(* IEC 61131-3 sources: std_i2980_v2.06_cp053/Source/IMM/ieccontrol/MoldGeneral (part 4) *)

(* ---- ABManualButton.pu ---- *)
(*
@h    ! WARNING !
@h    The Kemro K2 system (including software) only meets category B according to EN 954-1,
@h    thus it is not intended for usage in safety-relevant control applications in the field
@h    of personal safety (e.g. emergency stop).
@h    To implement potentially necessary safety-relevant control tasks, always use additional
@h    external safety devices that are intended for the particular purpose, and meet the necessary
@h    functional safety.
@h    For further information see EN 954-1 (EN ISO 13849-1) and/or the K2-x00 user manual, chapter
@h    "CE conformity, directives and standards".

react to manual buttons
find next target position when button is pressed

@FunctionID: S_FU_01_Mold1
*)

IMPORT_OVER_LISTFILE
 IS_LINKED
, cMoveFwd
, cMoveBwd
, cCompMoldHeightAuto
, cMoveBwdInterPos
, FBManualButton
, tsDeviceId
, tsInterCondList
, tsMoveData
, tyInstanceListArray
, tyInterCondBoolArray
, tMoveIdent
, FBCheckReady

END_IMPORT

ALGORITHM_BLOCK ABManualButton #DUMMY_EDIT_BLOCK

SYSTEM_VAR
 sv_bInitDone : BOOL;
 sv_DeviceId : tsDeviceId;
 sv_rMoldPosition : REAL;
 sv_FwdInterruptList : tsInterCondList (* list with interrupt positions for mold close *);
 sv_BwdInterruptList : tsInterCondList (* list with interrupt positions for mold open *);
 sv_MoveCloseInterPos : tsMoveData;
 sv_MoveOpenInterPos : tsMoveData;
 sv_bUseProgramSwitches : BOOL;
 sv_InstanceDataCloseInterPos : tyInstanceListArray;
 sv_InstanceDataOpenInterPos : tyInstanceListArray;
 sv_CloseInterPosProgInSequ : tyInterCondBoolArray (* information, which instances of mold close interpos movement are programmed in sequence  *);
 sv_OpenInterPosProgInSequ : tyInterCondBoolArray (* information, which instances of mold open interpos movement are programmed in sequence *);
END_VAR

SYSTEM_OBJECT
 PU_Task_7 : TASK;
END_OBJECT

VAR
 fbManualButton : FBManualButton;
 mpbAutoAdjustReady : REFTO BOOL;
END_VAR

ALGORITHM aGetNextCloseMovement

VAR_OUTPUT
 MoveId : tMoveIdent;
 iInstance : DINT;
END_VAR

VAR_TEMP
 i : DINT;
END_VAR
#BEGIN_EDIT_BLOCK
(**************************************** WARNING ********************************************
 *** The KEBA Kemro K2 System including software is not intended for safety control tasks! ***
 ***                       For further information see Comment tab!                        ***
 *********************************************************************************************)

MoveId := cMoveFwd;
iInstance := 1;

IF sv_bUseProgramSwitches THEN
   //get next target position from sv_FwdInterruptList
   FOR i := 1 TO sv_FwdInterruptList.iUsedElements DO
      IF (sv_FwdInterruptList.List[i].rTargetValue < sv_rMoldPosition) THEN
         iInstance := i;
         MoveId := cMoveFwdInterPos;
         RETURN;
      END_IF;
   END_FOR;
ELSE
   //sequence programmed by editor
   //-> check instance data to get next target position
   FOR i := 1 TO cMaxIntermediateConditions DO
      IF sv_CloseInterPosProgInSequ[i] AND sv_InstanceDataCloseInterPos[i].rTargetValue < sv_rMoldPosition THEN
         iInstance := i;
         MoveId := cMoveFwdInterPos;
         RETURN;
      END_IF;
   END_FOR;
END_IF;

;#END_EDIT_BLOCK END_ALGORITHM

ALGORITHM aGetNextOpenMovement

VAR_OUTPUT
 MoveId : tMoveIdent;
 iInstance : DINT;
END_VAR

VAR_TEMP
 i : DINT;
END_VAR
#BEGIN_EDIT_BLOCK
(**************************************** WARNING ********************************************
 *** The KEBA Kemro K2 System including software is not intended for safety control tasks! ***
 ***                       For further information see Comment tab!                        ***
 *********************************************************************************************)

MoveId := cMoveBwd;
iInstance := 1;

IF sv_bUseProgramSwitches THEN
   //get next target position from sv_BwdInterruptList
   FOR i := 1 TO sv_BwdInterruptList.iUsedElements DO
      IF (sv_BwdInterruptList.List[i].rTargetValue > sv_rMoldPosition) THEN
         iInstance := i;
         MoveId := cMoveBwdInterPos;
         RETURN;
      END_IF;
   END_FOR;
ELSE
   //sequence programmed by editor
   //-> check instance data to get next target position
   FOR i := 1 TO cMaxIntermediateConditions DO
      IF sv_OpenInterPosProgInSequ[i] AND sv_InstanceDataOpenInterPos[i].rTargetValue > sv_rMoldPosition THEN
         iInstance := i;
         MoveId := cMoveBwdInterPos;
         RETURN;
      END_IF;
   END_FOR;
END_IF;

;#END_EDIT_BLOCK END_ALGORITHM

ALGORITHM aButtonClose

VAR_INPUT
 bButtonClose : BOOL;
END_VAR

VAR
 MoveId : tMoveIdent;
 iIntermediateCond : DINT;
END_VAR
#BEGIN_EDIT_BLOCK
(**************************************** WARNING ********************************************
 *** The KEBA Kemro K2 System including software is not intended for safety control tasks! ***
 ***                       For further information see Comment tab!                        ***
 *********************************************************************************************)

IF mpbAutoAdjustReady <> EMPTY AND NOT mpbAutoAdjustReady^ THEN
    // auto mold adjust available and active -> ignore manual button
    RETURN;
END_IF;

IF bButtonClose THEN

   IF sv_MoveCloseInterPos.bProgrammedInSequence THEN
      //mold close movement to interpos programmed in sequence
      aGetNextCloseMovement(MoveId => MoveId,
                            iInstance => iIntermediateCond);
   ELSE
      //no interpos movement programmed
      MoveId := cMoveFwd;
      iIntermediateCond := 1;
   END_IF;

END_IF;

fbManualButton(bButton := bButtonClose, MoveId := MoveId, MoveDir := cMoveFwd, IntermediateCond := iIntermediateCond);

;#END_EDIT_BLOCK END_ALGORITHM

ALGORITHM aButtonOpen

VAR_INPUT
 bButtonOpen : BOOL;
END_VAR

VAR
 MoveId : tMoveIdent;
 iIntermediateCond : DINT;
END_VAR
#BEGIN_EDIT_BLOCK
(**************************************** WARNING ********************************************
 *** The KEBA Kemro K2 System including software is not intended for safety control tasks! ***
 ***                       For further information see Comment tab!                        ***
 *********************************************************************************************)

IF mpbAutoAdjustReady <> EMPTY AND NOT mpbAutoAdjustReady^ THEN
    // auto mold adjust available and active -> ignore manual button
    RETURN;
END_IF;

IF bButtonOpen THEN

   IF sv_MoveOpenInterPos.bProgrammedInSequence THEN
      //mold open movement to interpos programmed in sequence
      aGetNextOpenMovement(MoveId => MoveId,
                           iInstance => iIntermediateCond);
   ELSE
      //no interpos movement programmed
      MoveId := cMoveBwd;
      iIntermediateCond := 1;
   END_IF;

END_IF;

fbManualButton(bButton := bButtonOpen, MoveId := MoveId, MoveDir := cMoveBwd, IntermediateCond := iIntermediateCond);

;#END_EDIT_BLOCK END_ALGORITHM

POSTUPDATE_ALGORITHM pInitDone ON PU_Task_7(10) WITH sv_bInitDone

VAR
 fbCheckAutoAdjustReady : FBCheckReady;
 DeviceIdAutoAdjust : tsDeviceId;
END_VAR
#BEGIN_EDIT_BLOCK
(**************************************** WARNING ********************************************
 *** The KEBA Kemro K2 System including software is not intended for safety control tasks! ***
 ***                       For further information see Comment tab!                        ***
 *********************************************************************************************)

//get reference to ready flag of auto mold adjust function unit
DeviceIdAutoAdjust.CompId := cCompMoldHeightAuto;
DeviceIdAutoAdjust.IndexId := sv_DeviceId.IndexId;

fbCheckAutoAdjustReady(DeviceId := DeviceIdAutoAdjust);
mpbAutoAdjustReady := fbCheckAutoAdjustReady.pbReady;

;#END_EDIT_BLOCK END_ALGORITHM

END_ALGORITHM_BLOCK

#END_OF_IEC_PART

@Puma @IecEditor 6 97 @Pou 25
@@@BEG_Comment@@@
@h    ! WARNING !
@h    The Kemro K2 system (including software) only meets category B according to EN 954-1,
@h    thus it is not intended for usage in safety-relevant control applications in the field
@h    of personal safety (e.g. emergency stop).
@h    To implement potentially necessary safety-relevant control tasks, always use additional
@h    external safety devices that are intended for the particular purpose, and meet the necessary
@h    functional safety.
@h    For further information see EN 954-1 (EN ISO 13849-1) and/or the K2-x00 user manual, chapter
@h    "CE conformity, directives and standards".

react to manual buttons
find next target position when button is pressed

@FunctionID: S_FU_01_Mold1
@@@END_Comment@@@

@BEG_Contents

@BEG_Func
@RT(17)FuncTreeContainer
1
@Var @RT(9)IS_LINKED @RT(0) @T @T @DERIVED 0 @F @RT(22)KEBA_STANDARD_FUNCTION @F
@T
@BEG_Attrib
0 @RT(0) @RT(0)
@END_Attrib
1 1 @F @F @F @F

@END_Func

@BEG_Const
@RT(18)ConstTreeContainer
4
@Var @RT(8)cMoveFwd @RT(0) @T @F @DT @RT(4)DINT @RT(0) @T @T @BASIC 0 @F
@F @F
@T
@BEG_Attrib
0 @RT(2)12 @RT(16)movement forward
@END_Attrib
1 1 @F @F @F @F

@Var @RT(8)cMoveBwd @RT(0) @T @F @DT @RT(4)DINT @RT(0) @T @T @BASIC 0 @F
@F @F
@T
@BEG_Attrib
0 @RT(2)11 @RT(17)movement backward
@END_Attrib
1 1 @F @F @F @F

@Var @RT(19)cCompMoldHeightAuto @RT(0) @T @F @DT @RT(4)DINT @RT(0) @T @T @BASIC 0 @F
@F @F
@T
@BEG_Attrib
0 @RT(3)125 @RT(26)Component Auto Mold Height
@END_Attrib
1 1 @F @F @F @F

@Var @RT(16)cMoveBwdInterPos @RT(0) @T @F @DT @RT(4)DINT @RT(0) @T @T @BASIC 0 @F
@F @F
@T
@BEG_Attrib
0 @RT(2)16 @RT(38)move backward to intermediate position
@END_Attrib
1 1 @F @F @F @F

@END_Const

@BEG_Export

@BEG_Kind
@ALGORITHM_BLOCK @RT(14)ABManualButton @STRUCTURED_TEXT
@RT(0) @RT(0) @RT(0)
@END_Kind

@BEG_Dcl
@RT(16)DclTreeContainer
15
@Var @RT(9)PU_Task_7 @RT(0) @T @T @RENAMED 0 @T @T @DT @RT(4)TASK @RT(0) @T @T @BASIC 0 @F
@F @F
@T
@BEG_Attrib
3 @RT(0) @RT(0) @RT(0)
@END_Attrib
1 7 @F @F @F @F

@Var @RT(14)fbManualButton @RT(0) @T @T @DERIVED 0 @T @T @DT @RT(14)FBManualButton @RT(0) @T @T @UNKNOWN 0 @F
@F @F
@T
@BEG_Attrib
3 @RT(0) @RT(0) @RT(0)
@END_Attrib
1 0 @F @F @F @F

@Var @RT(12)sv_bInitDone @RT(0) @T @F @DT @RT(4)BOOL @RT(0) @T @T @BASIC 0 @F
@F @F
@T
@BEG_Attrib
3 @RT(0) @RT(0) @RT(0)
@END_Attrib
1 8 @F @F @F @F

@Var @RT(11)sv_DeviceId @RT(0) @T @T @DERIVED 0 @T @T @DT @RT(10)tsDeviceId @RT(0) @T @T @UNKNOWN 0 @F
@F @F
@T
@BEG_Attrib
3 @RT(0) @RT(0) @RT(0)
@END_Attrib
1 8 @F @F @F @F

@Var @RT(18)mpbAutoAdjustReady @RT(0) @T @T @REFTO 0 @T @DT @RT(4)BOOL @RT(0) @T @T @BASIC 0 @F
@F @F
@T
@BEG_Attrib
3 @RT(0) @RT(0) @RT(0)
@END_Attrib
1 0 @F @F @F @F

@Var @RT(16)sv_rMoldPosition @RT(0) @T @F @DT @RT(4)REAL @RT(0) @T @T @BASIC 0 @F
@F @F
@T
@BEG_Attrib
3 @RT(0) @RT(0) @RT(0)
@END_Attrib
1 8 @F @F @F @F

@Var @RT(19)sv_FwdInterruptList @RT(0) @T @T @DERIVED 0 @T @T @DT @RT(15)tsInterCondList @RT(0) @T @T @UNKNOWN 0 @F
@F @F
@T
@BEG_Attrib
3 @RT(0) @RT(44)list with interrupt positions for mold close @RT(0)
@END_Attrib
1 8 @F @F @F @F

@Var @RT(19)sv_BwdInterruptList @RT(0) @T @T @DERIVED 0 @T @T @DT @RT(15)tsInterCondList @RT(0) @T @T @UNKNOWN 0 @F
@F @F
@T
@BEG_Attrib
3 @RT(0) @RT(43)list with interrupt positions for mold open @RT(0)
@END_Attrib
1 8 @F @F @F @F

@Var @RT(20)sv_MoveCloseInterPos @RT(0) @T @T @DERIVED 0 @T @T @DT @RT(10)tsMoveData @RT(0) @T @T @UNKNOWN 0 @F
@F @F
@T
@BEG_Attrib
3 @RT(0) @RT(0) @RT(0)
@END_Attrib
1 8 @F @F @F @F

@Var @RT(19)sv_MoveOpenInterPos @RT(0) @T @T @DERIVED 0 @T @T @DT @RT(10)tsMoveData @RT(0) @T @T @UNKNOWN 0 @F
@F @F
@T
@BEG_Attrib
3 @RT(0) @RT(0) @RT(0)
@END_Attrib
1 8 @F @F @F @F

@Var @RT(22)sv_bUseProgramSwitches @RT(0) @T @F @DT @RT(4)BOOL @RT(0) @T @T @BASIC 0 @F
@F @F
@T
@BEG_Attrib
3 @RT(0) @RT(0) @RT(0)
@END_Attrib
1 8 @F @F @F @F

@Var @RT(28)sv_InstanceDataCloseInterPos @RT(0) @T @T @DERIVED 0 @T @T @DT @RT(19)tyInstanceListArray @RT(0) @T @T @UNKNOWN 0 @F
@F @F
@T
@BEG_Attrib
3 @RT(0) @RT(0) @RT(0)
@END_Attrib
1 8 @F @F @F @F

@Var @RT(27)sv_InstanceDataOpenInterPos @RT(0) @T @T @DERIVED 0 @T @T @DT @RT(19)tyInstanceListArray @RT(0) @T @T @UNKNOWN 0 @F
@F @F
@T
@BEG_Attrib
3 @RT(0) @RT(0) @RT(0)
@END_Attrib
1 8 @F @F @F @F

@Var @RT(26)sv_CloseInterPosProgInSequ @RT(0) @T @T @DERIVED 0 @T @T @DT @RT(20)tyInterCondBoolArray @RT(0) @T @T @UNKNOWN 0 @F
@F @F
@T
@BEG_Attrib
3 @RT(0) @RT(88)information, which instances of mold close interpos movement are programmed in sequence  @RT(0)
@END_Attrib
1 8 @F @F @F @F

@Var @RT(25)sv_OpenInterPosProgInSequ @RT(0) @T @T @DERIVED 0 @T @T @DT @RT(20)tyInterCondBoolArray @RT(0) @T @T @UNKNOWN 0 @F
@F @F
@T
@BEG_Attrib
3 @RT(0) @RT(86)information, which instances of mold open interpos movement are programmed in sequence @RT(0)
@END_Attrib
1 8 @F @F @F @F

@END_Dcl

@END_Export

@BEG_Body

5

@BEG_Export

@BEG_Algo
@ALGORITHM @RT(21)aGetNextCloseMovement @STRUCTURED_TEXT
@RT(0) @RT(0) @RT(0) @F @F
@END_Algo

@BEG_Dcl
@RT(16)DclTreeContainer
3
@Var @RT(6)MoveId @RT(0) @T @T @DERIVED 0 @T @T @DT @RT(10)tMoveIdent @RT(0) @T @T @UNKNOWN 0 @F
@F @F
@T
@BEG_Attrib
3 @RT(0) @RT(0) @RT(0)
@END_Attrib
1 3 @F @F @F @F

@Var @RT(9)iInstance @RT(0) @T @F @DT @RT(4)DINT @RT(0) @T @T @BASIC 0 @F
@F @F
@T
@BEG_Attrib
3 @RT(0) @RT(0) @RT(0)
@END_Attrib
1 3 @F @F @F @F

@Var @RT(1)i @RT(0) @T @F @DT @RT(4)DINT @RT(0) @T @T @BASIC 0 @F
@F @F
@T
@BEG_Attrib
3 @RT(0) @RT(0) @RT(0)
@END_Attrib
1 4 @F @F @F @F

@END_Dcl

@END_Export

@BEG_Export

@BEG_Algo
@ALGORITHM @RT(20)aGetNextOpenMovement @STRUCTURED_TEXT
@RT(0) @RT(0) @RT(0) @F @F
@END_Algo

@BEG_Dcl
@RT(16)DclTreeContainer
3
@Var @RT(6)MoveId @RT(0) @T @T @DERIVED 0 @T @T @DT @RT(10)tMoveIdent @RT(0) @T @T @UNKNOWN 0 @F
@F @F
@T
@BEG_Attrib
3 @RT(0) @RT(0) @RT(0)
@END_Attrib
1 3 @F @F @F @F

@Var @RT(9)iInstance @RT(0) @T @F @DT @RT(4)DINT @RT(0) @T @T @BASIC 0 @F
@F @F
@T
@BEG_Attrib
3 @RT(0) @RT(0) @RT(0)
@END_Attrib
1 3 @F @F @F @F

@Var @RT(1)i @RT(0) @T @F @DT @RT(4)DINT @RT(0) @T @T @BASIC 0 @F
@F @F
@T
@BEG_Attrib
3 @RT(0) @RT(0) @RT(0)
@END_Attrib
1 4 @F @F @F @F

@END_Dcl

@END_Export

@BEG_Export

@BEG_Algo
@ALGORITHM @RT(12)aButtonClose @STRUCTURED_TEXT
@RT(0) @RT(0) @RT(0) @F @F
@END_Algo

@BEG_Dcl
@RT(16)DclTreeContainer
3
@Var @RT(12)bButtonClose @RT(0) @T @F @DT @RT(4)BOOL @RT(0) @T @T @BASIC 0 @F
@F @F
@T
@BEG_Attrib
3 @RT(0) @RT(0) @RT(0)
@END_Attrib
1 1 @F @F @F @F

@Var @RT(6)MoveId @RT(0) @T @T @DERIVED 0 @T @T @DT @RT(10)tMoveIdent @RT(0) @T @T @UNKNOWN 0 @F
@F @F
@T
@BEG_Attrib
3 @RT(0) @RT(0) @RT(0)
@END_Attrib
1 0 @F @F @F @F

@Var @RT(17)iIntermediateCond @RT(0) @T @F @DT @RT(4)DINT @RT(0) @T @T @BASIC 0 @F
@F @F
@T
@BEG_Attrib
3 @RT(0) @RT(0) @RT(0)
@END_Attrib
1 0 @F @F @F @F

@END_Dcl

@END_Export

@BEG_Export

@BEG_Algo
@ALGORITHM @RT(11)aButtonOpen @STRUCTURED_TEXT
@RT(0) @RT(0) @RT(0) @F @F
@END_Algo

@BEG_Dcl
@RT(16)DclTreeContainer
3
@Var @RT(11)bButtonOpen @RT(0) @T @F @DT @RT(4)BOOL @RT(0) @T @T @BASIC 0 @F
@F @F
@T
@BEG_Attrib
3 @RT(0) @RT(0) @RT(0)
@END_Attrib
1 1 @F @F @F @F

@Var @RT(6)MoveId @RT(0) @T @T @DERIVED 0 @T @T @DT @RT(10)tMoveIdent @RT(0) @T @T @UNKNOWN 0 @F
@F @F
@T
@BEG_Attrib
3 @RT(0) @RT(0) @RT(0)
@END_Attrib
1 0 @F @F @F @F

@Var @RT(17)iIntermediateCond @RT(0) @T @F @DT @RT(4)DINT @RT(0) @T @T @BASIC 0 @F
@F @F
@T
@BEG_Attrib
3 @RT(0) @RT(0) @RT(0)
@END_Attrib
1 0 @F @F @F @F

@END_Dcl

@END_Export

@BEG_Export

@BEG_Algo
@POSTUPDATE_ALGORITHM @RT(9)pInitDone @STRUCTURED_TEXT
@RT(0) @RT(12)sv_bInitDone @RT(13)PU_Task_7(10) @F @F
@END_Algo

@BEG_Dcl
@RT(16)DclTreeContainer
2
@Var @RT(22)fbCheckAutoAdjustReady @RT(0) @T @T @DERIVED 0 @T @T @DT @RT(12)FBCheckReady @RT(0) @T @T @UNKNOWN 0 @F
@F @F
@T
@BEG_Attrib
3 @RT(0) @RT(0) @RT(0)
@END_Attrib
1 0 @F @F @F @F

@Var @RT(18)DeviceIdAutoAdjust @RT(0) @T @T @DERIVED 0 @T @T @DT @RT(10)tsDeviceId @RT(0) @T @T @UNKNOWN 0 @F
@F @F
@T
@BEG_Attrib
3 @RT(0) @RT(0) @RT(0)
@END_Attrib
1 0 @F @F @F @F

@END_Dcl

@END_Export

@BEG_Body
@TL(31)
(**************************************** WARNING ********************************************
 *** The KEBA Kemro K2 System including software is not intended for safety control tasks! ***
 ***                       For further information see Comment tab!                        ***
 *********************************************************************************************)

MoveId := cMoveFwd;
iInstance := 1;

IF sv_bUseProgramSwitches THEN
   //get next target position from sv_FwdInterruptList
   FOR i := 1 TO sv_FwdInterruptList.iUsedElements DO
      IF (sv_FwdInterruptList.List[i].rTargetValue < sv_rMoldPosition) THEN
         iInstance := i;
         MoveId := cMoveFwdInterPos;
         RETURN;
      END_IF;
   END_FOR;
ELSE
   //sequence programmed by editor
   //-> check instance data to get next target position
   FOR i := 1 TO cMaxIntermediateConditions DO
      IF sv_CloseInterPosProgInSequ[i] AND sv_InstanceDataCloseInterPos[i].rTargetValue < sv_rMoldPosition THEN
         iInstance := i;
         MoveId := cMoveFwdInterPos;
         RETURN;
      END_IF;
   END_FOR;
END_IF;

@END_Body

@@@BEG_Comment@@@
@TL(0)

@@@END_Comment@@@

@BEG_Body
@TL(31)
(**************************************** WARNING ********************************************
 *** The KEBA Kemro K2 System including software is not intended for safety control tasks! ***
 ***                       For further information see Comment tab!                        ***
 *********************************************************************************************)

MoveId := cMoveBwd;
iInstance := 1;

IF sv_bUseProgramSwitches THEN
   //get next target position from sv_BwdInterruptList
   FOR i := 1 TO sv_BwdInterruptList.iUsedElements DO
      IF (sv_BwdInterruptList.List[i].rTargetValue > sv_rMoldPosition) THEN
         iInstance := i;
         MoveId := cMoveBwdInterPos;
         RETURN;
      END_IF;
   END_FOR;
ELSE
   //sequence programmed by editor
   //-> check instance data to get next target position
   FOR i := 1 TO cMaxIntermediateConditions DO
      IF sv_OpenInterPosProgInSequ[i] AND sv_InstanceDataOpenInterPos[i].rTargetValue > sv_rMoldPosition THEN
         iInstance := i;
         MoveId := cMoveBwdInterPos;
         RETURN;
      END_IF;
   END_FOR;
END_IF;

@END_Body

@@@BEG_Comment@@@
@TL(0)

@@@END_Comment@@@

@BEG_Body
@TL(26)
(**************************************** WARNING ********************************************
 *** The KEBA Kemro K2 System including software is not intended for safety control tasks! ***
 ***                       For further information see Comment tab!                        ***
 *********************************************************************************************)

IF mpbAutoAdjustReady <> EMPTY AND NOT mpbAutoAdjustReady^ THEN
    // auto mold adjust available and active -> ignore manual button
    RETURN;
END_IF;

IF bButtonClose THEN

   IF sv_MoveCloseInterPos.bProgrammedInSequence THEN
      //mold close movement to interpos programmed in sequence
      aGetNextCloseMovement(MoveId => MoveId,
                            iInstance => iIntermediateCond);
   ELSE
      //no interpos movement programmed
      MoveId := cMoveFwd;
      iIntermediateCond := 1;
   END_IF;

END_IF;

fbManualButton(bButton := bButtonClose, MoveId := MoveId, MoveDir := cMoveFwd, IntermediateCond := iIntermediateCond);

@END_Body

@@@BEG_Comment@@@
@TL(0)

@@@END_Comment@@@

@BEG_Body
@TL(27)
(**************************************** WARNING ********************************************
 *** The KEBA Kemro K2 System including software is not intended for safety control tasks! ***
 ***                       For further information see Comment tab!                        ***
 *********************************************************************************************)

IF mpbAutoAdjustReady <> EMPTY AND NOT mpbAutoAdjustReady^ THEN
    // auto mold adjust available and active -> ignore manual button
    RETURN;
END_IF;

IF bButtonOpen THEN

   IF sv_MoveOpenInterPos.bProgrammedInSequence THEN
      //mold open movement to interpos programmed in sequence
      aGetNextOpenMovement(MoveId => MoveId,
                           iInstance => iIntermediateCond);
   ELSE
      //no interpos movement programmed
      MoveId := cMoveBwd;
      iIntermediateCond := 1;
   END_IF;

END_IF;

fbManualButton(bButton := bButtonOpen, MoveId := MoveId, MoveDir := cMoveBwd, IntermediateCond := iIntermediateCond);

@END_Body

@@@BEG_Comment@@@
@TL(0)

@@@END_Comment@@@

@BEG_Body
@TL(13)
(**************************************** WARNING ********************************************
 *** The KEBA Kemro K2 System including software is not intended for safety control tasks! ***
 ***                       For further information see Comment tab!                        ***
 *********************************************************************************************)

//get reference to ready flag of auto mold adjust function unit
DeviceIdAutoAdjust.CompId := cCompMoldHeightAuto;
DeviceIdAutoAdjust.IndexId := sv_DeviceId.IndexId;

fbCheckAutoAdjustReady(DeviceId := DeviceIdAutoAdjust);
mpbAutoAdjustReady := fbCheckAutoAdjustReady.pbReady;

@END_Body

@@@BEG_Comment@@@
@TL(0)

@@@END_Comment@@@
@END_Body

@END_Contents

(* ---- ABMoldProtection.pu ---- *)
(*
@h    ! WARNING !
@h    The Kemro K2 system (including software) only meets category B according to EN 954-1,
@h    thus it is not intended for usage in safety-relevant control applications in the field
@h    of personal safety (e.g. emergency stop).
@h    To implement potentially necessary safety-relevant control tasks, always use additional
@h    external safety devices that are intended for the particular purpose, and meet the necessary
@h    functional safety.
@h    For further information see EN 954-1 (EN ISO 13849-1) and/or the K2-x00 user manual, chapter
@h    "CE conformity, directives and standards".

This algorithm block is used for mold protect detection

function:
When movement is active and in protect stage a timer is started.
If movement stops in protect stage (button released) and continues again then the timer will also continue.
If timer is equal the allowed time (dProtectTime) a protection error is detected and
all mold fwd movements are locked automatically.
Furthermore a protect event (evProtect) is sent.
After pressing the alarm confirm button, the mold fwd movements will be unlocked.

@FunctionID: S_KPIEC_ALAOP_02
*)

IMPORT_OVER_LISTFILE
 cCompMold
, tevAlarmConfirm
, tevProtect
, tsDeviceId
, ALARM_EVENT
, tnOperationMode
, tnLockUnlock
, FBLockUnlock
, KAPPL_VisProfile
, TON
, R_TRIG
, tevProtectData
, ALARM_EVENT_DATA
, tevAlarmConfirmData

END_IMPORT

ALGORITHM_BLOCK ABMoldProtection #DUMMY_EDIT_BLOCK

SYSTEM_VAR
 sv_DeviceId : tsDeviceId;
 sv_bInitDone : BOOL;
 sv_iActMoldProtectRetry : DINT;
 sv_iSetMoldProtectRetry : DINT;
 sv_bOpenAfterProtect : BOOL;
 sv_OperationMode : tnOperationMode;
END_VAR

SYSTEM_OBJECT
 erMoldProtection : ALARM;
 EV_Task_7 : TASK;
 evAlarmConfirm : tevAlarmConfirm;
 evProtect : tevProtect;
 evAlarmAutoManual : ALARM_EVENT;
END_OBJECT

(*
This algorithm locks/unlocks all mold fwd movements
*)

ALGORITHM aLockUnlock

VAR_INPUT
 nMode : tnLockUnlock;
END_VAR

VAR
 bInitDone : BOOL;
 fbLockUnlock : FBLockUnlock;
END_VAR
#BEGIN_EDIT_BLOCK
(**************************************** WARNING ********************************************
 *** The KEBA Kemro K2 System including software is not intended for safety control tasks! ***
 ***                       For further information see Comment tab!                        ***
 *********************************************************************************************)

IF NOT sv_bInitDone THEN
   RETURN;
END_IF;

IF NOT bInitDone THEN
   fbLockUnlock.DeviceId.CompId := cCompMold;
   fbLockUnlock.DeviceId.IndexId := 1;
   fbLockUnlock.MoveDir := cMoveFwd;
   fbLockUnlock.MoveId := cMoveAll;
   fbLockUnlock.Alarm.AlarmId := erMoldProtection;
   bInitDone := TRUE;
END_IF;

fbLockUnlock.Mode := nMode;

//lock all mold fwd movements
fbLockUnlock();

;#END_EDIT_BLOCK END_ALGORITHM

(*
In this algorithm the detection of protect erros is done
*)

ALGORITHM aRun

VAR_INPUT
 bMovementActive : BOOL (* activate detection *);
 rActPosition : REAL (* actual mold position *);
 pVisProfile : REFTO KAPPL_VisProfile (* pointer to mold close profile *);
 dProtectTime : TIME (* set mold protect time *);
END_VAR

VAR_OUTPUT
 dActTime : TIME (* elapsed protect time *);
 bMoldProtectError : BOOL (* mold protect error detected *);
END_VAR

VAR
 fbTonProtect : TON;
 fbRTrigActive : R_TRIG;
 rProtectStartPos : REAL (* startposition of mold protect *);
 rProtectEndPos : REAL (* endposition of mold protect *);
 dLastProtectTime : TIME;
 dAllowedProtectTime : TIME;
 evProtectData : tevProtectData;
 evAlarmAutoManualData : ALARM_EVENT_DATA;
 bProtectOnce : BOOL;
 dummy : DINT;
END_VAR
#BEGIN_EDIT_BLOCK
(**************************************** WARNING ********************************************
 *** The KEBA Kemro K2 System including software is not intended for safety control tasks! ***
 ***                       For further information see Comment tab!                        ***
 *********************************************************************************************)

rProtectStartPos := pVisProfile^.Profile.Points[(pVisProfile^.Profile.iNoOfPoints-1)].rStartPos;
rProtectEndPos := pVisProfile^.Profile.Points[pVisProfile^.Profile.iNoOfPoints].rStartPos;

fbRTrigActive(CLK := bMovementActive);
IF fbRTrigActive.Q THEN
    IF (rActPosition < rProtectStartPos) AND (rActPosition > rProtectEndPos) AND NOT bMoldProtectError THEN
       //movement started and mold already in mold protect area and no protect error occured at last mold move
       dLastProtectTime := dActTime; //save elapsed time from last mold movement and continue timer
    ELSE
       //mold out of protect area at start of movement or mold protect error occured last time
       dLastProtectTime := t#0.0s;
    END_IF;

    dAllowedProtectTime := dProtectTime - dLastProtectTime;
    fbTonProtect(IN := FALSE);
    bProtectOnce := FALSE;

END_IF;

IF bMovementActive THEN
   IF (rActPosition < rProtectStartPos) AND rActPosition > rProtectEndPos THEN
      // mold in mold protection area
      fbTonProtect(IN := TRUE,
                   PT := dAllowedProtectTime);
      dActTime := fbTonProtect.ET + dLastProtectTime;
   ELSE
      //mold outside mold protect area
      fbTonProtect(IN := FALSE);
   END_IF;

   bMoldProtectError := fbTonProtect.Q;

   IF fbTonProtect.Q AND NOT bProtectOnce THEN
      dummy := Print('send mold protect event');

      IF (sv_OperationMode > nManual) AND sv_bOpenAfterProtect AND (sv_iActMoldProtectRetry < sv_iSetMoldProtectRetry) THEN
         //only switch opmode, no alarm or buzzer
         SET_EVENT(evAlarmAutoManual, evAlarmAutoManualData);
      ELSE
          //lock all mold fwd movements
         aLockUnlock(nMode := nLockAbort);
      END_IF;

      //send protect event
      evProtectData.DeviceIdSender := sv_DeviceId;
      evProtectData.DeviceIdReceiver.CompId := cCompMold;
      evProtectData.DeviceIdReceiver.IndexId := 1;
      SET_EVENT(evProtect, evProtectData);
   END_IF;

   bProtectOnce := fbTonProtect.Q;
END_IF;

;#END_EDIT_BLOCK END_ALGORITHM

(*
This event algorithm reacts on pressing the alarm confirm button.
After alarm confirmation all mold fwd movements are unlocked
*)

EVENT_ALGORITHM evaAlarmConfirm ON EV_Task_7 WITH evAlarmConfirm

VAR_INPUT
 evAlarmConfirmData : tevAlarmConfirmData;
END_VAR
#BEGIN_EDIT_BLOCK
(**************************************** WARNING ********************************************
 *** The KEBA Kemro K2 System including software is not intended for safety control tasks! ***
 ***                       For further information see Comment tab!                        ***
 *********************************************************************************************)

//unlock all mold fwd movements when alarm confirm button is pressed
aLockUnlock(nMode := nUnlock);

;#END_EDIT_BLOCK END_ALGORITHM

END_ALGORITHM_BLOCK

#END_OF_IEC_PART

@Puma @IecEditor 6 68 @Pou 25
@@@BEG_Comment@@@
@h    ! WARNING !
@h    The Kemro K2 system (including software) only meets category B according to EN 954-1,
@h    thus it is not intended for usage in safety-relevant control applications in the field
@h    of personal safety (e.g. emergency stop).
@h    To implement potentially necessary safety-relevant control tasks, always use additional
@h    external safety devices that are intended for the particular purpose, and meet the necessary
@h    functional safety.
@h    For further information see EN 954-1 (EN ISO 13849-1) and/or the K2-x00 user manual, chapter
@h    "CE conformity, directives and standards".

This algorithm block is used for mold protect detection

function:
When movement is active and in protect stage a timer is started.
If movement stops in protect stage (button released) and continues again then the timer will also continue.
If timer is equal the allowed time (dProtectTime) a protection error is detected and
all mold fwd movements are locked automatically.
Furthermore a protect event (evProtect) is sent.
After pressing the alarm confirm button, the mold fwd movements will be unlocked.

@FunctionID: S_KPIEC_ALAOP_02
@@@END_Comment@@@

@BEG_Contents

@BEG_Func
@RT(17)FuncTreeContainer
0
@END_Func

@BEG_Const
@RT(18)ConstTreeContainer
1
@Var @RT(9)cCompMold @RT(0) @T @F @DT @RT(4)DINT @RT(0) @T @T @BASIC 0 @F
@F @F
@T
@BEG_Attrib
0 @RT(3)101 @RT(14)Component Mold
@END_Attrib
1 1 @F @F @F @F

@END_Const

@BEG_Export

@BEG_Kind
@ALGORITHM_BLOCK @RT(16)ABMoldProtection @STRUCTURED_TEXT
@RT(0) @RT(0) @RT(0)
@END_Kind

@BEG_Dcl
@RT(16)DclTreeContainer
11
@Var @RT(16)erMoldProtection @RT(0) @T @F @DT @RT(5)ALARM @RT(0) @T @T @BASIC 0 @F
@F @F
@T
@BEG_Attrib
3 @RT(0) @RT(0) @RT(0)
@END_Attrib
1 7 @F @F @F @F

@Var @RT(9)EV_Task_7 @RT(0) @T @F @DT @RT(4)TASK @RT(0) @T @T @BASIC 0 @F
@F @F
@T
@BEG_Attrib
3 @RT(0) @RT(0) @RT(0)
@END_Attrib
1 7 @F @F @F @F

@Var @RT(14)evAlarmConfirm @RT(0) @T @T @RENAMED 0 @T @T @DT @RT(15)tevAlarmConfirm @RT(0) @T @T @UNKNOWN 0 @F
@F @F
@T
@BEG_Attrib
3 @RT(0) @RT(0) @RT(0)
@END_Attrib
1 7 @F @F @F @F

@Var @RT(9)evProtect @RT(0) @T @T @DERIVED 0 @T @T @DT @RT(10)tevProtect @RT(0) @T @T @UNKNOWN 0 @F
@F @F
@T
@BEG_Attrib
3 @RT(0) @RT(0) @RT(0)
@END_Attrib
1 7 @F @F @F @F

@Var @RT(11)sv_DeviceId @RT(0) @T @T @DERIVED 0 @T @T @DT @RT(10)tsDeviceId @RT(0) @T @T @UNKNOWN 0 @F
@F @F
@T
@BEG_Attrib
3 @RT(0) @RT(0) @RT(0)
@END_Attrib
1 8 @F @F @F @F

@Var @RT(12)sv_bInitDone @RT(0) @T @T @RENAMED 0 @T @T @DT @RT(4)BOOL @RT(0) @T @T @BASIC 0 @F
@F @F
@T
@BEG_Attrib
3 @RT(0) @RT(0) @RT(0)
@END_Attrib
1 8 @F @F @F @F

@Var @RT(23)sv_iActMoldProtectRetry @RT(0) @T @F @DT @RT(4)DINT @RT(0) @T @T @BASIC 0 @F
@F @F
@T
@BEG_Attrib
3 @RT(0) @RT(0) @RT(0)
@END_Attrib
1 8 @F @F @F @F

@Var @RT(23)sv_iSetMoldProtectRetry @RT(0) @T @F @DT @RT(4)DINT @RT(0) @T @T @BASIC 0 @F
@F @F
@T
@BEG_Attrib
3 @RT(0) @RT(0) @RT(0)
@END_Attrib
1 8 @F @F @F @F

@Var @RT(17)evAlarmAutoManual @RT(0) @T @T @RENAMED 0 @T @T @DT @RT(11)ALARM_EVENT @RT(0) @T @T @UNKNOWN 0 @F
@F @F
@T
@BEG_Attrib
3 @RT(0) @RT(0) @RT(0)
@END_Attrib
1 7 @F @F @F @F

@Var @RT(20)sv_bOpenAfterProtect @RT(0) @T @F @DT @RT(4)BOOL @RT(0) @T @T @BASIC 0 @F
@F @F
@T
@BEG_Attrib
3 @RT(0) @RT(0) @RT(0)
@END_Attrib
1 8 @F @F @F @F

@Var @RT(16)sv_OperationMode @RT(0) @T @T @DERIVED 0 @F @RT(15)tnOperationMode @F
@T
@BEG_Attrib
3 @RT(0) @RT(0) @RT(0)
@END_Attrib
1 8 @F @F @F @F

@END_Dcl

@END_Export

@BEG_Body

3

@BEG_Export

@BEG_Algo
@ALGORITHM @RT(11)aLockUnlock @STRUCTURED_TEXT
@RT(0) @RT(0) @RT(0) @F @F
@END_Algo

@BEG_Dcl
@RT(16)DclTreeContainer
3
@Var @RT(5)nMode @RT(0) @T @T @DERIVED 0 @T @T @DT @RT(12)tnLockUnlock @RT(0) @T @T @UNKNOWN 0 @F
@F @F
@T
@BEG_Attrib
3 @RT(0) @RT(0) @RT(0)
@END_Attrib
1 1 @F @F @F @F

@Var @RT(9)bInitDone @RT(0) @T @F @DT @RT(4)BOOL @RT(0) @T @T @BASIC 0 @F
@F @F
@T
@BEG_Attrib
3 @RT(0) @RT(0) @RT(0)
@END_Attrib
1 0 @F @F @F @F

@Var @RT(12)fbLockUnlock @RT(0) @T @T @DERIVED 0 @T @T @DT @RT(12)FBLockUnlock @RT(0) @T @T @UNKNOWN 0 @F
@F @F
@T
@BEG_Attrib
3 @RT(0) @RT(0) @RT(0)
@END_Attrib
1 0 @F @F @F @F

@END_Dcl

@END_Export

@BEG_Export

@BEG_Algo
@ALGORITHM @RT(4)aRun @STRUCTURED_TEXT
@RT(0) @RT(0) @RT(0) @F @F
@END_Algo

@BEG_Dcl
@RT(16)DclTreeContainer
16
@Var @RT(15)bMovementActive @RT(0) @T @F @DT @RT(4)BOOL @RT(0) @T @T @BASIC 0 @F
@F @F
@T
@BEG_Attrib
3 @RT(0) @RT(18)activate detection @RT(0)
@END_Attrib
1 1 @F @F @F @F

@Var @RT(12)rActPosition @RT(0) @T @F @DT @RT(4)REAL @RT(0) @T @T @BASIC 0 @F
@F @F
@T
@BEG_Attrib
3 @RT(0) @RT(20)actual mold position @RT(0)
@END_Attrib
1 1 @F @F @F @F

@Var @RT(11)pVisProfile @RT(0) @T @T @REFTO 0 @F @DERIVED 0 @T @T @DT @RT(16)KAPPL_VisProfile @RT(0) @T @T @UNKNOWN 0 @F
@F @F
@T
@BEG_Attrib
3 @RT(0) @RT(29)pointer to mold close profile @RT(0)
@END_Attrib
1 1 @F @F @F @F

@Var @RT(12)dProtectTime @RT(0) @T @F @DT @RT(4)TIME @RT(0) @T @T @BASIC 0 @F
@F @F
@T
@BEG_Attrib
3 @RT(0) @RT(21)set mold protect time @RT(0)
@END_Attrib
1 1 @F @F @F @F

@Var @RT(8)dActTime @RT(0) @T @F @DT @RT(4)TIME @RT(0) @T @T @BASIC 0 @F
@F @F
@T
@BEG_Attrib
3 @RT(0) @RT(20)elapsed protect time @RT(0)
@END_Attrib
1 3 @F @F @F @F

@Var @RT(17)bMoldProtectError @RT(0) @T @F @DT @RT(4)BOOL @RT(0) @T @T @BASIC 0 @F
@F @F
@T
@BEG_Attrib
3 @RT(0) @RT(27)mold protect error detected @RT(0)
@END_Attrib
1 3 @F @F @F @F

@Var @RT(12)fbTonProtect @RT(0) @T @T @DERIVED 0 @T @T @DT @RT(3)TON @RT(0) @T @T @UNKNOWN 0 @F
@F @F
@T
@BEG_Attrib
3 @RT(0) @RT(0) @RT(0)
@END_Attrib
1 0 @F @F @F @F

@Var @RT(13)fbRTrigActive @RT(0) @T @T @DERIVED 0 @T @T @DT @RT(6)R_TRIG @RT(0) @T @T @UNKNOWN 0 @F
@F @F
@T
@BEG_Attrib
3 @RT(0) @RT(0) @RT(0)
@END_Attrib
1 0 @F @F @F @F

@Var @RT(16)rProtectStartPos @RT(0) @T @F @DT @RT(4)REAL @RT(0) @T @T @BASIC 0 @F
@F @F
@T
@BEG_Attrib
3 @RT(0) @RT(29)startposition of mold protect @RT(0)
@END_Attrib
1 0 @F @F @F @F

@Var @RT(14)rProtectEndPos @RT(0) @T @F @DT @RT(4)REAL @RT(0) @T @T @BASIC 0 @F
@F @F
@T
@BEG_Attrib
3 @RT(0) @RT(27)endposition of mold protect @RT(0)
@END_Attrib
1 0 @F @F @F @F

@Var @RT(16)dLastProtectTime @RT(0) @T @F @DT @RT(4)TIME @RT(0) @T @T @BASIC 0 @F
@F @F
@T
@BEG_Attrib
3 @RT(0) @RT(0) @RT(0)
@END_Attrib
1 0 @F @F @F @F

@Var @RT(19)dAllowedProtectTime @RT(0) @T @F @DT @RT(4)TIME @RT(0) @T @T @BASIC 0 @F
@F @F
@T
@BEG_Attrib
3 @RT(0) @RT(0) @RT(0)
@END_Attrib
1 0 @F @F @F @F

@Var @RT(13)evProtectData @RT(0) @T @T @DERIVED 0 @T @T @DT @RT(14)tevProtectData @RT(0) @T @T @UNKNOWN 0 @F
@F @F
@T
@BEG_Attrib
3 @RT(0) @RT(0) @RT(0)
@END_Attrib
1 0 @F @F @F @F

@Var @RT(21)evAlarmAutoManualData @RT(0) @T @T @DERIVED 0 @T @T @DT @RT(16)ALARM_EVENT_DATA @RT(0) @T @T @UNKNOWN 0 @F
@F @F
@T
@BEG_Attrib
3 @RT(0) @RT(0) @RT(0)
@END_Attrib
1 0 @F @F @F @F

@Var @RT(12)bProtectOnce @RT(0) @T @F @DT @RT(4)BOOL @RT(0) @T @T @BASIC 0 @F
@F @F
@T
@BEG_Attrib
3 @RT(0) @RT(0) @RT(0)
@END_Attrib
1 0 @F @F @F @F

@Var @RT(5)dummy @RT(0) @T @F @DT @RT(4)DINT @RT(0) @T @T @BASIC 0 @F
@F @F
@T
@BEG_Attrib
3 @RT(0) @RT(0) @RT(0)
@END_Attrib
1 0 @F @F @F @F

@END_Dcl

@END_Export

@BEG_Export

@BEG_Algo
@EVENT_ALGORITHM @RT(15)evaAlarmConfirm @STRUCTURED_TEXT
@RT(0) @RT(14)evAlarmConfirm @RT(9)EV_Task_7 @F @F
@END_Algo

@BEG_Dcl
@RT(16)DclTreeContainer
1
@Var @RT(18)evAlarmConfirmData @RT(0) @T @T @DERIVED 0 @T @T @DT @RT(19)tevAlarmConfirmData @RT(0) @T @T @UNKNOWN 0 @F
@F @F
@T
@BEG_Attrib
3 @RT(0) @RT(0) @RT(0)
@END_Attrib
1 1 @F @F @F @F

@END_Dcl

@END_Export

@BEG_Body
@TL(23)
(**************************************** WARNING ********************************************
 *** The KEBA Kemro K2 System including software is not intended for safety control tasks! ***
 ***                       For further information see Comment tab!                        ***
 *********************************************************************************************)

IF NOT sv_bInitDone THEN
   RETURN;
END_IF;

IF NOT bInitDone THEN
   fbLockUnlock.DeviceId.CompId := cCompMold;
   fbLockUnlock.DeviceId.IndexId := 1;
   fbLockUnlock.MoveDir := cMoveFwd;
   fbLockUnlock.MoveId := cMoveAll;
   fbLockUnlock.Alarm.AlarmId := erMoldProtection;
   bInitDone := TRUE;
END_IF;

fbLockUnlock.Mode := nMode;

//lock all mold fwd movements
fbLockUnlock();

@END_Body

@@@BEG_Comment@@@
@TL(1)
This algorithm locks/unlocks all mold fwd movements
@@@END_Comment@@@

@BEG_Body
@TL(58)
(**************************************** WARNING ********************************************
 *** The KEBA Kemro K2 System including software is not intended for safety control tasks! ***
 ***                       For further information see Comment tab!                        ***
 *********************************************************************************************)

rProtectStartPos := pVisProfile^.Profile.Points[(pVisProfile^.Profile.iNoOfPoints-1)].rStartPos;
rProtectEndPos := pVisProfile^.Profile.Points[pVisProfile^.Profile.iNoOfPoints].rStartPos;

fbRTrigActive(CLK := bMovementActive);
IF fbRTrigActive.Q THEN
    IF (rActPosition < rProtectStartPos) AND (rActPosition > rProtectEndPos) AND NOT bMoldProtectError THEN
       //movement started and mold already in mold protect area and no protect error occured at last mold move
       dLastProtectTime := dActTime; //save elapsed time from last mold movement and continue timer
    ELSE
       //mold out of protect area at start of movement or mold protect error occured last time
       dLastProtectTime := t#0.0s;
    END_IF;

    dAllowedProtectTime := dProtectTime - dLastProtectTime;
    fbTonProtect(IN := FALSE);
    bProtectOnce := FALSE;

END_IF;

IF bMovementActive THEN
   IF (rActPosition < rProtectStartPos) AND rActPosition > rProtectEndPos THEN
      // mold in mold protection area
      fbTonProtect(IN := TRUE,
                   PT := dAllowedProtectTime);
      dActTime := fbTonProtect.ET + dLastProtectTime;
   ELSE
      //mold outside mold protect area
      fbTonProtect(IN := FALSE);
   END_IF;

   bMoldProtectError := fbTonProtect.Q;

   IF fbTonProtect.Q AND NOT bProtectOnce THEN
      dummy := Print('send mold protect event');

      IF (sv_OperationMode > nManual) AND sv_bOpenAfterProtect AND (sv_iActMoldProtectRetry < sv_iSetMoldProtectRetry) THEN
         //only switch opmode, no alarm or buzzer
         SET_EVENT(evAlarmAutoManual, evAlarmAutoManualData);
      ELSE
          //lock all mold fwd movements
         aLockUnlock(nMode := nLockAbort);
      END_IF;

      //send protect event
      evProtectData.DeviceIdSender := sv_DeviceId;
      evProtectData.DeviceIdReceiver.CompId := cCompMold;
      evProtectData.DeviceIdReceiver.IndexId := 1;
      SET_EVENT(evProtect, evProtectData);
   END_IF;

   bProtectOnce := fbTonProtect.Q;
END_IF;

@END_Body

@@@BEG_Comment@@@
@TL(1)
In this algorithm the detection of protect erros is done
@@@END_Comment@@@

@BEG_Body
@TL(9)
(**************************************** WARNING ********************************************
 *** The KEBA Kemro K2 System including software is not intended for safety control tasks! ***
 ***                       For further information see Comment tab!                        ***
 *********************************************************************************************)

//unlock all mold fwd movements when alarm confirm button is pressed
aLockUnlock(nMode := nUnlock);

@END_Body

@@@BEG_Comment@@@
@TL(2)
This event algorithm reacts on pressing the alarm confirm button.
After alarm confirmation all mold fwd movements are unlocked
@@@END_Comment@@@
@END_Body

@END_Contents
